// SIMATIC S7-200 project (STEP 7-Micro/WIN), CPU 222 CN REL 02.01

ORGANIZATION_BLOCK 主程序:OB1
TITLE=我手写了一个带加速功能的步进电机控制程序，供有需要的人参考。
// 在主程序中，首先通过系统运行状态检测和电机运行标志位判断运行条件，只有当系统运行状态为真且电机运行标志位为假时，重置步进电机使能输出并调用子程序，确保系统就绪。随后，主程序调用子程序配置步进电机的运行参数。当步进电机脉冲计数达到1时，置位步进电机状态指示，反映电机运行状态；当步进电机脉冲计数大于等于2时，将其重置为0，保持计数准确。
// 子程序负责设置步进电机的运行参数。步进电机控制模式配置被设置为特定值，步进电机速度设置被设为固定值，步进电机目标脉冲数被设为限定值，确保电机按预期运行。子程序通过相关参数配置加速阶段。子程序通过相关参数配置减速阶段。子程序通过相关参数配置恒速阶段，确保运行平稳。最后，子程序启用中断和脉冲输出，开始电机运动。
// 中断程序在每次脉冲触发时，将步进电机脉冲计数增加1，实时更新电机位置。
BEGIN
Network 1 // 网络标题
// 网络注释
LD     SM0.1
LD     M0.1
EU
OLD
R      Q0.0, 1
CALL   SBR_0:SBR0
Network 2
LDB=   VB10, 1
=      Q0.1
Network 3
LDB>=  VB10, 2
MOVB   0, VB10
END_ORGANIZATION_BLOCK

SUBROUTINE_BLOCK SBR_0:SBR0
TITLE=子程序注释
BEGIN
Network 1 // 网络标题
// 网络注释
LD     SM0.0
MOVB   16#A0, SMB67
MOVW   100, SMW168
MOVB   3, VB100
Network 2
LD     SM0.0
MOVW   1000, VW101
MOVW   -1, VW103
MOVD   876, VD105
Network 3
LD     SM0.0
MOVW   125, VW117
MOVW   0, VW119
MOVD   300000, VD121
Network 4
LD     SM0.0
MOVW   1000, VW125
MOVW   1, VW127
MOVD   876, VD129
Network 5
LD     SM0.0
ATCH   INT_0:INT0, 19
ENI
PLS    0
END_SUBROUTINE_BLOCK

INTERRUPT_BLOCK INT_0:INT0
TITLE=中断程序注释
BEGIN
Network 1 // 网络标题
// 网络注释
LD     SM0.0
INCB   VB10
END_INTERRUPT_BLOCK
